# EPICS substitutions: PSI/iocVxWorks.subs
file iocRTOS.template
{
pattern { IOCNAME , SYS_MBUF_FLNK     }
	{ "$(IOC)"  , "$(IOC):CLUST_1_0_0"}
}

file iocVxWorksOnly.template
{
pattern { IOCNAME , DAT_MBUF_FLNK     }
	{ "$(IOC)"  , "$(IOC):CLUST_0_0_0"}
}

file iocCluster.template
{
#                   Pool   Size
pattern { IOCNAME ,  P   ,  S   , TYPE , FLNK               }
# Data Pool
	{ "$(IOC)"  ,  0   ,  0   , DAT  , "$(IOC):CLUST_0_1_0" }
	{ "$(IOC)"  ,  0   ,  1   , DAT  , "$(IOC):CLUST_0_2_0" }
	{ "$(IOC)"  ,  0   ,  2   , DAT  , "$(IOC):CLUST_0_3_0" }
	{ "$(IOC)"  ,  0   ,  3   , DAT  , "$(IOC):CLUST_0_4_0" }
	{ "$(IOC)"  ,  0   ,  4   , DAT  , "$(IOC):CLUST_0_5_0" }
	{ "$(IOC)"  ,  0   ,  5   , DAT  , "$(IOC):CLUST_0_6_0" }
	{ "$(IOC)"  ,  0   ,  6   , DAT  , "$(IOC):CLUST_0_7_0" }
	{ "$(IOC)"  ,  0   ,  7   , DAT  , ""                 }
# System Pool
	{ "$(IOC)"  ,  1   ,  0   , SYS  , "$(IOC):CLUST_1_1_0" }
	{ "$(IOC)"  ,  1   ,  1   , SYS  , "$(IOC):CLUST_1_2_0" }
	{ "$(IOC)"  ,  1   ,  2   , SYS  , "$(IOC):CLUST_1_3_0" }
	{ "$(IOC)"  ,  1   ,  3   , SYS  , "$(IOC):CLUST_1_4_0" }
	{ "$(IOC)"  ,  1   ,  4   , SYS  , "$(IOC):CLUST_1_5_0" }
	{ "$(IOC)"  ,  1   ,  5   , SYS  , "$(IOC):CLUST_1_6_0" }
	{ "$(IOC)"  ,  1   ,  6   , SYS  , "$(IOC):CLUST_1_7_0" }
	{ "$(IOC)"  ,  1   ,  7   , SYS  , ""                 }
}

file iocEnvVar.template
{
pattern { IOCNAME, ENVNAME           , ENVVAR                       , ENVTYPE}
	{ "$(IOC)" , TIMEZONE        , TIMEZONE                     , env    }
}
